FUNCTION_BLOCK Thomas_Object EXTENDS TcoCore.TcoObject
VAR_INPUT
	_frank : AKid_Object(THIS^);
	_andrew : AKid_Object(THIS^);
	_christina : AKid_Object(THIS^);
	_gianna : AKid_Object(THIS^);
END_VAR

END_FUNCTION_BLOCK

(* stored: Version 1.1.0.1, ProductVersion 3.1.4024.6
   POU Thomas_Object: Id {69d01a44-cebd-0fff-162d-7a59f62e3932}, SpecialFunc None *)
